// TwinCAT 3 PLC project HALT
// ProgramVersion: 3.1.4024.0
// libraries:
//   Tc2_Standard, * (Beckhoff Automation GmbH)
//   Tc2_System, * (Beckhoff Automation GmbH)
//   Tc3_Module, * (Beckhoff Automation GmbH)
//   TcUnit, * (www.tcunit.org)
//   VisuSymbols,3.5.10.0,System
// project tree:
//   DUTs/ stLimit.TcDUT
//   / GlobalTextList.TcGTLO, PlcTask.TcTTO, Visualization Manager.TcVMO (not stored)
//   POUs/ FCheckVariabel.TcPOU, HPU_BLOCK.TcPOU, MAIN.TcPOU, Safety_Block.TcPOU, VFD_BLOCK.TcPOU
//   VISUs/ Visualization.TcVIS
// real-time tasks:
//   TASK PlcTask: cycle T#10ms, priority 20, ADS port 350
// I/O:
//   DEVICE Device 1 (EtherCAT), AmsNetId 5.24.235.67.2.1
//     Term 16 (EK1200)
//   DEVICE Device 4 (NOV-DP-RAM)
// variable links:
//   HALT/HALT Instance <-> Device 1 (EtherCAT)/Term 16 (EK1200)/Term 10 (EL2004)
//     PlcTask Outputs/MAIN.fbVfdBlock.bOnOffVfd1ControlRelaySeven <-> Channel 1/Output
//     PlcTask Outputs/MAIN.fbVfdBlock.bOnOffVfd3ControlRelayTen <-> Channel 4/Output
//     PlcTask Outputs/MAIN.fbVfdBlock.bReverseVfd1ControlRelayEight <-> Channel 2/Output
//   HALT/HALT Instance <-> Device 1 (EtherCAT)/Term 16 (EK1200)/Term 12 (EL3356-0010)
//     PlcTask Inputs/MAIN.iForceMeasurement <-> RMB Value (INT32)/Value
//   HALT/HALT Instance <-> Device 1 (EtherCAT)/Term 16 (EK1200)/Term 2 (EL3122)
//     PlcTask Inputs/MAIN.iPositionMeasurment <-> AI Standard Channel 1/Value
//   HALT/HALT Instance <-> Device 1 (EtherCAT)/Term 16 (EK1200)/Term 3 (EL3152)
//     PlcTask Inputs/MAIN.iPerssureMeasurementPort1 <-> AI Standard Channel 1/Value
//     PlcTask Inputs/MAIN.iPerssureMeasurementPort2 <-> AI Standard Channel 2/Value
//   HALT/HALT Instance <-> Device 1 (EtherCAT)/Term 16 (EK1200)/Term 4 (EL3202)
//     PlcTask Inputs/MAIN.iTemperatureMeasurementPort1 <-> RTD Inputs Channel 1/Value
//     PlcTask Inputs/MAIN.iTemperatureMeasurementPort2 <-> RTD Inputs Channel 2/Value
//   HALT/HALT Instance <-> Device 1 (EtherCAT)/Term 16 (EK1200)/Term 5 (EL4002)
//     PlcTask Outputs/MAIN.fbVfdBlock.aiThe10VoltagesSignalForTheSpeedReferenceControlToTheVfD1 <-> AO Outputs Channel 1/Analog output
//   HALT/HALT Instance <-> Device 1 (EtherCAT)/Term 16 (EK1200)/Term 6 (EL2022)
//     PlcTask Outputs/MAIN.fbHpuBlock.bHpuMotorControlRelayTwo <-> Channel 2/Output
//   HALT/HALT Instance <-> Device 1 (EtherCAT)/Term 16 (EK1200)/Term 7 (EL1004)
//     PlcTask Inputs/MAIN.fbSafetyBlock.bSafetyDetectionRelay <-> Channel 1/Input
//   HALT/HALT Instance <-> Device 1 (EtherCAT)/Term 16 (EK1200)/Term 8 (EL1004)
//     PlcTask Inputs/MAIN.fbSafetyBlock.bLimitSwitchLeft <-> Channel 4/Input
//     PlcTask Inputs/MAIN.fbSafetyBlock.bLimitSwitchRight <-> Channel 2/Input
//   HALT/HALT Instance <-> Device 1 (EtherCAT)/Term 16 (EK1200)/Term 9 (EL2004)
//     PlcTask Outputs/MAIN.fbHpuBlock.bHpuValveControlRelayFive <-> Channel 4/Output
//     PlcTask Outputs/MAIN.fbHpuBlock.bPneumaticBreakValveControlRelaySix <-> Channel 3/Output
//     PlcTask Outputs/MAIN.fbSafetyBlock.bSafetyCircuitRelayFour <-> Channel 2/Output
//     PlcTask Outputs/MAIN.fbSafetyBlock.bSafetyCircuitRelayThree <-> Channel 1/Output

CONFIGURATION HALT
    RESOURCE PLC ON TwinCAT3
        TASK PlcTask(INTERVAL := T#10ms, PRIORITY := 20);
        PROGRAM MAIN WITH PlcTask : MAIN;
    END_RESOURCE
END_CONFIGURATION

// ---- DUTs/stLimit.TcDUT
TYPE stLimit  :
STRUCT
    rMinimumValue : REAL;      // Lower bound for the REAL value to be tested 
    rMaxiumValue : REAL;      // Upper bound for the REAL value to be tested 
    bValueMustBe : BOOL;      // Whtere if the varirable BOOL must be TRUE or FALSE
END_STRUCT
END_TYPE

// ---- POUs/MAIN.TcPOU
PROGRAM MAIN
VAR
	// Measurabel Variabels 
    iTemperatureMeasurementPort1   AT %I* : INT;   // temperature port 1
    iTemperatureMeasurementPort2   AT %I* : INT;   // temperature port 2
    iPerssureMeasurementPort1  AT %I* : INT;   // pressure port 1
    iPerssureMeasurementPort2  AT %I* : INT;   // pressure port 2
    iPositionMeasurment     AT %I* : INT;   // position
    iForceMeasurement   AT %I* : DINT;   // force
	
	// Readable Variabels
    rTemperatureReadable1 : REAL;   // temperature port 1
    rTemperatureReadable2 : REAL;   // temperature port 2
    rPerssureReadable1 : REAL;   // pressure port 1
    rPerssureReadable2 : REAL;   // pressure port 2
    rPositionReadable : REAL;   // position
    rForceReadable : REAL;   // force
	
	// Relay Variabels: // 
	// bSafetyCircuitRelayThree				    AT %Q* : BOOL; // This is the on/off variable for the third relay in the system, which can break the safety circuit
	// bSafetyCircuitRelayFour					AT %Q* : BOOL; // This is the on/off variable for the fourth relay in the system, which can break the safety circuit
	// bHpuValveControlRelayFive				AT %Q* : BOOL; // This is the on/off variable for the fifth relay in the system, which is used to turn on and off the HPU valve
	// bPneumaticBreakValveControlRelaySix		AT %Q* : BOOL; // This is the on/off variable for the sixth relay in the system, which is used to turn on and off the pneumatic break valve
	// bOnOffVfd1ControlRelaySeven				AT %Q* : BOOL; // This is the on/off variable for the seventh relay in the system, which is used to turn on and off the VFD 1
	// bReverseVfd1ControlRelayEight			AT %Q* : BOOL; // This is the change‑direction variable for the eighth relay in the system, which is used to set the direction of the VFD 1

	// System Variabels: //
	// Time - DT - Data and time  
	// OperationalSystemValue - BOOL - This is a indicating value to indicate if the system is operational or not
	
	// Measuuerbal Parameteres: // 
	// iTemperatureMeasurementPort1 AT %I* : INT;
	// iTemperatureMeasurementPort2 AT %I* : INT;
	// PerssureMeasurementPort1 - INT - 
	// PerssureMeasurementPort2 - INT - 
	// ForceMeasurement - INT - 
	// iPositionMeasurment AT %I* : INT; 
	// iVelocityMeasurment AT %I* : INT ; 

	
	// LimitSwitch Variabels: // 
	// LimitSwitchRight - BOOL - 
	// LimitSwitchLeft - BOOL - 
	
	// VFD Variabels: // 
	// VfdOn - BOOL - 
	// VfdOff - BOOL - 
	// VfdClockwiseRotation - BOOL - 
	// VfdCounterClockwiseRotation - BOOL - 
	// VfdPositionReference - INT - 
	// VfdSpeedReference - INT - 
	
	// Set Parameters: //
	iTestMode AT %I* : INT;
	rLongStrockDistanceSet  AT %I* : REAL; 
	rLongStrockVelocitySet  AT %I* : REAL; 
	rMicroStrockAngularSpeedSet AT %I* : REAL; 
	rOilTemperatureSet AT %I* : REAL; 
	rOilPressureSet AT %I* : REAL; 
	
	bSTOP AT %I* : BOOL := TRUE; 
	
	fbSafetyBlock : Safety_Block;
	fbVfdBlock : VFD_BLOCK;
	fbHpuBlock : HPU_BLOCK;
END_VAR

// Make and scale the data readable
rTemperatureReadable1 := INT_TO_REAL(iTemperatureMeasurementPort1) / 10;
rTemperatureReadable2 := INT_TO_REAL(iTemperatureMeasurementPort1) / 10;
rPerssureReadable1 := INT_TO_REAL(iPerssureMeasurementPort1) / 32768.0 * 400.0;
rPerssureReadable2 := INT_TO_REAL(iPerssureMeasurementPort2) / 32768.0 * 400.0;
rPositionReadable := (INT_TO_REAL(iPositionMeasurment) / 32768) * 1000;
rForceReadable := DINT_TO_REAL(iForceMeasurement);


// Pass measured values to the safety block
fbSafetyBlock.rTemperature1 := rTemperatureReadable1;
fbSafetyBlock.rTemperature2 := rTemperatureReadable2;
fbSafetyBlock.rPressure1    := rPerssureReadable1 ;
fbSafetyBlock.rPressure2    := rPerssureReadable1 ;
fbSafetyBlock.rPosition     := rPositionReadable;
fbSafetyBlock.rForce        := rForceReadable;
fbSafetyBlock.STOP          := bSTOP;

// Execute the safety block
fbSafetyBlock();

fbVfdBlock();
fbHpuBlock();

// 2004 1 1 = R3
// 2004 1 2 = R4
// 2004 1 3 = R6 
// 2004 1 4 = R5
// 2004 2 1 = R7
// 2004 2 2 = R8
// 2004 2 4 = R9

END_PROGRAM

// ---- POUs/Safety_Block.TcPOU
FUNCTION_BLOCK Safety_Block
VAR_INPUT
    //--- Limit‑switch signals ---------------------------------
    bLimitSwitchRight   AT %I* : BOOL;   // right‑hand limit switch
    bLimitSwitchLeft    AT %I* : BOOL;   // left‑hand limit switch
    bSafetyDetectionRelay AT %I* : BOOL; // safety relay detection
    bHmiActivationBottom AT %I* : BOOL;  // HMI activation button

    //--- Measured values (passed as inputs) --------------------
    rTemperature1       : REAL;           // temperature port 1
    rTemperature2       : REAL;           // temperature port 2
    rPressure1          : REAL;           // pressure port 1
    rPressure2          : REAL;           // pressure port 2
    rPosition           : REAL;           // position
    rForce              : REAL;           // force
	
	STOP 				: BOOL; // 

    //--- Limit definitions ------------------------------------
    stTemperatureLimit1 : stLimit := (rMinimumValue:=0.0, rMaxiumValue:=120.0, bValueMustBe:=FALSE);
    stTemperatureLimit2 : stLimit := (rMinimumValue:=0.0, rMaxiumValue:=120.0, bValueMustBe:=FALSE);
    stPressureLimit1    : stLimit := (rMinimumValue:=95.0,  rMaxiumValue:=110.0, bValueMustBe:=FALSE);
    stPressureLimit2    : stLimit := (rMinimumValue:=95.0,  rMaxiumValue:=110.0, bValueMustBe:=FALSE);
    stPositionLimit     : stLimit := (rMinimumValue:=0.0,   rMaxiumValue:=1000.0, bValueMustBe:=FALSE);
    stForceLimit        : stLimit := (rMinimumValue:=0.0,   rMaxiumValue:=1000.0, bValueMustBe:=FALSE);
    stSafetyLimit       : stLimit := (rMinimumValue:=0.0,   rMaxiumValue:=0.0,   bValueMustBe:=TRUE);   // must be TRUE
END_VAR

VAR_OUTPUT
    bAllOk               AT %Q* : BOOL;          // all limits satisfied
    bSafetyCircuitRelayThree AT %Q* : BOOL := FALSE;      // third safety relay
    bSafetyCircuitRelayFour  AT %Q* : BOOL := FALSE;      // fourth safety relay
	bSystemIsUpAndRuning AT %Q* : BOOL; // 
END_VAR

VAR
    //--- Results of individual checks -------------------------
    bOkTemperature1      : BOOL;
    bOkTemperature2      : BOOL;
    bOkPressure1         : BOOL;
    bOkPressure2         : BOOL;
    bOkPosition          : BOOL;
    bOkForce             : BOOL;
    bOkLimitSwitchRight  : BOOL;
    bOkLimitSwitchLeft   : BOOL;
END_VAR

// Temperature checks
bOkTemperature1 := FCheckVariabel(rTemperature1, stTemperatureLimit1);
bOkTemperature2 := FCheckVariabel(rTemperature2, stTemperatureLimit2);

// Pressure checks
bOkPressure1 := FCheckVariabel(rPressure1, stPressureLimit1);
bOkPressure2 := FCheckVariabel(rPressure2, stPressureLimit2);

// Position check
bOkPosition := FCheckVariabel(rPosition, stPositionLimit);

// Force check
bOkForce := FCheckVariabel(rForce, stForceLimit);

// Limit‑switch checks (BOOL → REAL, because FCheckVariabel expects REAL)
bOkLimitSwitchRight := FCheckVariabel(BOOL_TO_REAL(bLimitSwitchRight), stSafetyLimit);
bOkLimitSwitchLeft  := FCheckVariabel(BOOL_TO_REAL(bLimitSwitchLeft),  stSafetyLimit);

// Overall OK status – every single check must be TRUE
bAllOk := bOkTemperature1
	   AND bOkTemperature2
//	   AND bOkPressure1
//	   AND bOkPressure2
	   AND bOkPosition
	   AND bOkForce
	   AND bOkLimitSwitchRight
	   AND bOkLimitSwitchLeft
	   AND bHmiActivationBottom;


IF NOT STOP THEN 
	bSystemIsUpAndRuning := FALSE;
	bSafetyCircuitRelayThree := FALSE;
	bSafetyCircuitRelayFour  := FALSE;
ELSE
	// Activate the safety relays only when all limits are satisfied
	IF bAllOk THEN
		bSafetyCircuitRelayThree := TRUE;
		bSafetyCircuitRelayFour  := TRUE;
	ELSE
		bSafetyCircuitRelayThree := FALSE;
		bSafetyCircuitRelayFour  := FALSE;
	END_IF

	IF bAllOk AND bSafetyDetectionRelay THEN 
		bSystemIsUpAndRuning := TRUE;
	ELSE
		bSystemIsUpAndRuning := FALSE;
	END_IF
END_IF

END_FUNCTION_BLOCK

// ---- POUs/FCheckVariabel.TcPOU
FUNCTION FCheckVariabel :BOOL
VAR_INPUT
    rValue   : REAL;      // The accuel value (can also be a BOOL, that the bool is either 0/1)
    stLimit   : stLimit;    // limit ‑ definition for this variable
END_VAR

// If it is a BOOL, we ignore min / max and only look at bValueMustBe
IF (stLimit.rMinimumValue = 0.0) AND (stLimit.rMaxiumValue = 0.0) THEN
	FCheckVariabel := (rValue <> 0.0) = stLimit.bValueMustBe;   // value <> 0.0 = TRUE hvis BOOL er TRUE
ELSE
	// otherwise it is a REAL that must be within min / max
	FCheckVariabel := (rValue >= stLimit.rMinimumValue) AND (rValue <= stLimit.rMaxiumValue );
END_IF;

END_FUNCTION

// ---- POUs/VFD_BLOCK.TcPOU
FUNCTION_BLOCK VFD_BLOCK
VAR_INPUT
	rPositionMeasurment : REAL;
	rVfdPositionReference : REAL; 
	rSet AT %I* : REAL;
END_VAR
VAR_OUTPUT
	bOnOffVfd1ControlRelaySeven				AT %Q* : BOOL; // This is the on/off variable for the seventh relay in the system, which is used to turn on and off the VFD 1
	bReverseVfd1ControlRelayEight			AT %Q* : BOOL; // This is the change‑direction variable for the eighth relay in the system, which is used to set the direction of the VFD 1
	bOnOffVfd3ControlRelayTen				AT %Q* : BOOL; // This is the on/off variable for the tenth relay in the system, which is used to turn on and off the VFD 2
	aiThe10VoltagesSignalForTheSpeedReferenceControlToTheVfD1 AT %Q* : INT;
	
END_VAR
VAR
	bEnable : BOOL;

END_VAR
VAR_TEMP
	fScale : REAL;
END_VAR

bEnable := TRUE;

IF bEnable THEN

   (* Clamp setpoint *)
   IF rSet > 100.0 THEN
      rSet := 100.0;
   ELSIF rSet < 0.0 THEN
      rSet := 0.0;
   END_IF;

   (* Scale output *)
   fScale := rSet / 100.0;
   aiThe10VoltagesSignalForTheSpeedReferenceControlToTheVfD1 := REAL_TO_INT(fScale * 32767.0);


ELSE

   aiThe10VoltagesSignalForTheSpeedReferenceControlToTheVfD1 := 0;

END_IF;

END_FUNCTION_BLOCK

// ---- POUs/HPU_BLOCK.TcPOU
FUNCTION_BLOCK HPU_BLOCK
VAR_INPUT 
END_VAR
VAR_OUTPUT
	bHpuMotorControlRelayTwo				AT %Q* : BOOL := FALSE; // This is the on/off variable for the second relay in the system, which is used to turn on and off the HPU motor
	bHpuValveControlRelayFive				AT %Q* : BOOL := FALSE; // This is the on/off variable for the fifth relay in the system, which is used to turn on and off the HPU valve
	bPneumaticBreakValveControlRelaySix		AT %Q* : BOOL := FALSE; // This is the on/off variable for the sixth relay in the system, which is used to turn on and off the pneumatic break valve
	
END_VAR
VAR
END_VAR


IF  MAIN.rPerssureReadable1 > 110 THEN 
	bHpuMotorControlRelayTwo := FALSE;
	bHpuValveControlRelayFive := FALSE;
END_IF

END_FUNCTION_BLOCK

// ---- GlobalTextList.TcGTLO
TEXTLIST GlobalTextList
  916 = '%r'
  219 = 'Actication'
  364 = 'Activate the system'
  728 = 'asda'
  909 = 'asdad'
  351 = 'Force on the rod: %0.00f N'
  319 = 'Force on the rod: &0.00f N'
  153 = 'Force on the rod: &f0.0f N'
  604 = 'GroupBox'
  718 = 'HPU Contactor'
  501 = 'HPU Motor '
  954 = 'HPU Valve'
  212 = 'Long Strock '
  885 = 'Long Strock - backwards'
  799 = 'Long Strock - Backwards'
  888 = 'Long Strock - Forwards'
  766 = 'Manually Control '
  191 = 'Measuret Data'
  892 = 'Measurments'
  590 = 'Micro Strock'
  982 = 'Operation'
  594 = 'Pneumatic Valve'
  294 = 'Position of the rod: %0.00f mm'
  841 = 'Position of the rod: %0.0f mm'
  847 = 'Power'
  878 = 'Pressure of port 1: %0.00f Bar'
  317 = 'Pressure of port 1: %0.0f Bar'
  98 = 'Pressure of port 2: %0.00f Bar'
  471 = 'Pressure of port 2: %0.0f Bar'
  633 = 'Rember to press the REST bottom after the activate bottum'
  733 = 'Set Parameters'
  929 = 'Set the Long Strock Distance '
  530 = 'Set the Long Strock Distance (0 - 1000 mm) '
  330 = 'Set the Long Strock Velocity'
  195 = 'Set the Long Strock Velocity (0 - 300 mm/s)'
  371 = 'Set the Long Strock Velocity (0-300 mm/s)'
  368 = 'Set the longstrock mode:'
  643 = 'Set the micro strock (0 - 5 Hz )'
  591 = 'Set the micro strock (0 - 5 Hz)'
  580 = 'Set the micro strock (0-5 Hz'
  403 = 'Set the micro strock Hz'
  775 = 'Set the oli pressure'
  348 = 'Set The Oli Pressure'
  95 = 'Set The Oli Pressure (0 - 120 Bar)'
  726 = 'Set The Oli Temperature'
  354 = 'Set The Oli Temperature (0 - 120 C)'
  107 = 'Set the Test Mode'
  46 = 'Set the Test Mode (1-5)'
  174 = 'Sikkerhed 1'
  358 = 'Sikkerhed 2'
  778 = 'STOP'
  920 = 'STOP Operations'
  585 = 'Temprature of port 1: %0.00f C'
  746 = 'Temprature of port 1: %0.0f C'
  372 = 'Temprature of port 2: %0.00f C'
  694 = 'Temprature of port 2: %0.0f C'
  455 = 'The LED is on when the system in operational'
END_TEXTLIST

// ---- VISUs/Visualization.TcVIS
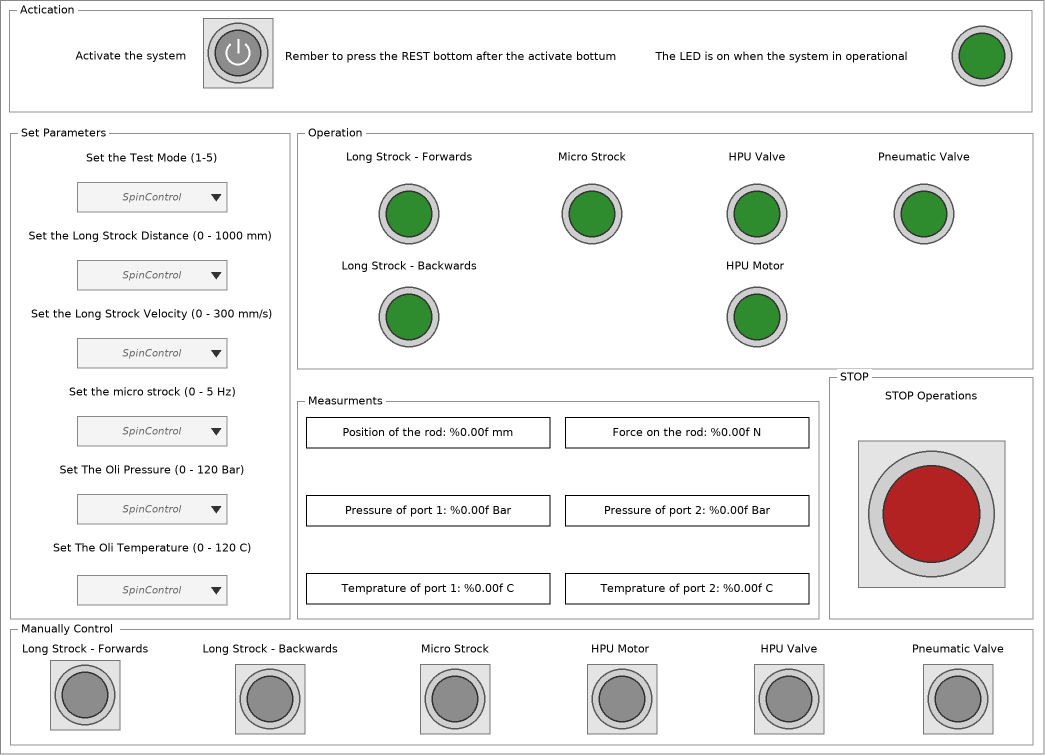
VISUALIZATION Visualization  // 1045x755
    GroupBox (9,2 1023x110), "Actication"
        Label (38,26 168x56), "Activate the system"
        Label (276,40 331x29), "Rember to press the REST bottom after the activate bottum"
        Lamp1 (938,19 70x70), variable: MAIN.fbSafetyBlock.bSystemIsUpAndRuning, style: Lamp-Lamp1-Green
        Label (607,40 331x29), "The LED is on when the system in operational"
        PowerSwitch (194,16 70x70), variable: MAIN.fbSafetyBlock.bHmiActivationBottom, behaviour: TOGGLE, style: Switch-PowerSwitch-Gray
    GroupBox (10,125 280x494), "Set Parameters"
        SpinControl (67,57 150x30), variable: MAIN.iTestMode
            OnMouseClick: write the text variable via Edit, min 0, max 5, format %i
        SpinControl (67,291 150x30), variable: MAIN.rMicroStrockAngularSpeedSet
            p1653691745: 0.1
            OnMouseClick: write the text variable via Edit, min 0, max 1000, format %r
        SpinControl (67,369 150x30), variable: MAIN.rOilPressureSet
            OnMouseClick: write the text variable via Edit, min 0, max 120, format %r
        SpinControl (67,450 150x30), variable: MAIN.rOilTemperatureSet
            OnMouseClick: write the text variable via Edit, min 0, max 120, format %r
        Label (67,18 150x30), "Set the Test Mode (1-5)"
        Label (50,252 185x30), "Set the micro strock (0 - 5 Hz)"
        Label (28,408 229x30), "Set The Oli Temperature (0 - 120 C)"
        Label (39,330 206x30), "Set The Oli Pressure (0 - 120 Bar)"
        SpinControl (67,135 150x30), variable: MAIN.rLongStrockDistanceSet
            OnMouseClick: write the text variable via Edit, min 0, max 1000, format %i
        Label (11,96 262x30), "Set the Long Strock Distance (0 - 1000 mm)"
        SpinControl (67,213 150x30), variable: MAIN.fbVfdBlock.rSet
            OnMouseClick: write the text variable via Edit, min 0, max 300, format %i
        Label (13,174 258x30), "Set the Long Strock Velocity (0 - 300 mm/s)"
    GroupBox (297,393 522x226), "Measurments"
        RoundedRectangle (9,180 244x31), "Temprature of port 1: %0.00f C", text variable: MAIN.rTemperatureReadable1
        RoundedRectangle (268,180 244x31), "Temprature of port 2: %0.00f C", text variable: MAIN.rTemperatureReadable2
        RoundedRectangle (9,102 244x31), "Pressure of port 1: %0.00f Bar", text variable: MAIN.rPerssureReadable1
        RoundedRectangle (268,102 244x31), "Pressure of port 2: %0.00f Bar", text variable: MAIN.rPerssureReadable2
        RoundedRectangle (268,24 244x31), "Force on the rod: %0.00f N", text variable: MAIN.rForceReadable
        RoundedRectangle (9,24 244x31), "Position of the rod: %0.00f mm", text variable: MAIN.rPositionReadable
    GroupBox (297,125 736x244), "Operation"
        Lamp1 (425,54 70x70), variable: MAIN.fbHpuBlock.bHpuValveControlRelayFive, style: Lamp-Lamp1-Green
        Lamp1 (425,157 70x70), variable: MAIN.fbHpuBlock.bHpuMotorControlRelayTwo, style: Lamp-Lamp1-Green
        Label (385,126 150x30), "HPU Motor"
        Label (385,17 150x30), "HPU Valve"
        Lamp1 (592,54 70x70), style: Lamp-Lamp1-Green
        Label (552,17 150x30), "Pneumatic Valve"
        Lamp1 (260,54 70x70), style: Lamp-Lamp1-Green
        Label (220,17 150x30), "Micro Strock"
        Lamp1 (77,54 70x70), style: Lamp-Lamp1-Green
        Label (37,17 150x30), "Long Strock - Forwards"
        Lamp1 (77,157 70x70), style: Lamp-Lamp1-Green
        Label (19,126 186x30), "Long Strock - Backwards"
    GroupBox (829,369 204x250), "STOP"
        Label (27,12 150x30), "STOP Operations"
        PushSwitchLed (29,63 147x164), variable: MAIN.bSTOP, behaviour: TOGGLE, style: Switch-PushSwitchLed-Red
    GroupBox (10,621 1023x124), "Manually Control"
        Label (0,13 150x30), "Long Strock - Forwards"
        Label (167,13 186x30), "Long Strock - Backwards"
        Label (370,13 150x30), "Micro Strock"
        Label (537,13 150x30), "HPU Motor"
        Label (704,13 150x30), "HPU Valve"
        Label (873,13 150x30), "Pneumatic Valve"
        PushSwitchLed (40,39 70x70), variable: MAIN.fbVfdBlock.bOnOffVfd1ControlRelaySeven, behaviour: TOGGLE, style: Switch-PushSwitchLed-Gray
        PushSwitchLed (225,43 70x70), behaviour: TAP, style: Switch-PushSwitchLed-Gray
        PushSwitchLed (410,43 70x70), behaviour: TAP, style: Switch-PushSwitchLed-Gray
        PushSwitchLed (577,43 70x70), variable: MAIN.fbHpuBlock.bHpuMotorControlRelayTwo, behaviour: TAP, style: Switch-PushSwitchLed-Gray
        PushSwitchLed (744,43 70x70), variable: MAIN.fbHpuBlock.bHpuValveControlRelayFive, behaviour: TOGGLE, style: Switch-PushSwitchLed-Gray
        PushSwitchLed (913,43 70x70), behaviour: TAP, style: Switch-PushSwitchLed-Gray
END_VISUALIZATION
